Staubli VAL3: robotPlanner.pgx

public program robotPlanner(num& x_nFileID[], num& x_ndForceTorque[], pointRx& x_pdPointPos[], num& x_ndPointVel[], num& x_ndPointAccel[], jointRx& x_jdJointPos[], num& x_ndJointVel[], num& x_ndJointAccel[])
begin

  //====================  从文件输入机器人运动规划所期望的数据（Force/Motion State） ====================

  //---------- 从外部文件输入更新机器人运动规划的期望力和位置（待后期补充） ----------
  //期望的机器人与环境交互作用力Force
  //$fileGet(x_nFileID[3],x_ndForceTorque[0],6)

  //期望的机器人的运动状态Motion State
  //笛卡尔空间内（Cartesian Space）
  //$fileGet(x_nFileID[4],x_pdPointPos[0],6)
  //$fileGet(x_nFileID[4],x_ndPointVel[0],6)
  //$fileGet(x_nFileID[4],x_ndPointAccel[0],6)

  //关节空间内（Joint Space）
  //$fileGet(x_nFileID[5],x_jdJointPos[0],6)
  //$fileGet(x_nFileID[5],x_ndJointVel[0],6)
  //$fileGet(x_nFileID[5],x_ndJointAccel[0],6)


  //---------- 当前假定期望力为零，期望位置保持不变（注意单位换算，当前使用MKS） ----------
  //期望的机器人与环境交互作用力Force（N）
  x_ndForceTorque[0]=0
  x_ndForceTorque[1]=0
  x_ndForceTorque[2]=0
  x_ndForceTorque[3]=0
  x_ndForceTorque[4]=0
  x_ndForceTorque[5]=0


  //期望的机器人的运动状态Motion State（m,m/s,m/s^2;°,°/s,°/s^2）
  //笛卡尔空间内（Cartesian Space）
  //加速度
  x_ndPointAccel=0

  //速度
  x_ndPointVel=0

  //位置和姿态
  x_pdPointPos=pNowPointPos

  //关节空间内（Joint Space）
  //加速度
  //x_ndJointAccel=0

  //速度
  //x_ndJointVel=0

  //位置
  //x_jdJointPos=jNowJointPos

end
